FUNCTION_BLOCK FB_SelfTest IMPLEMENTS I_State
VAR_INPUT
	(* Pointer to the ATM Machine*)
	pATM_Machine	: POINTER TO FB_ATM_Machine;
END_VAR
VAR_OUTPUT
END_VAR
VAR
END_VAR

METHOD Cancel : BOOL
END_METHOD

METHOD Card_Ejected : BOOL
END_METHOD

METHOD Card_Inserted : BOOL
END_METHOD

PROPERTY Description : E_StateDescription
GET
Description := E_StateDescription.SelfTest;
END_GET
END_PROPERTY

METHOD Failure : BOOL
ADSLOGSTR(ADSLOG_MSGTYPE_LOG, 'System Test Fail, going to Out of Service', '');
pATM_Machine^.SetState(pATM_Machine^.OutOfServiceState);
END_METHOD

METHOD FB_Init : BOOL
VAR_INPUT
	(* if TRUE, the retain variables are initialized (warm start / cold start)*)
	bInitRetains	: BOOL;
	(* if TRUE, the instance afterwards gets moved into the copy code (online change)*)
	bInCopyCode	: BOOL;
	(* Pointer to the ATM Machine*)
	pATM_Machine	: POINTER TO FB_ATM_Machine;
END_VAR
THIS^.pATM_Machine := pATM_Machine;
END_METHOD

METHOD Op : BOOL
END_METHOD

METHOD Service : BOOL
END_METHOD

METHOD SystemTest_OK : BOOL
ADSLOGSTR(ADSLOG_MSGTYPE_LOG, 'System Test Pass, going to Idel', '');
pATM_Machine^.SetState(pATM_Machine^.IdleState);
END_METHOD

METHOD Turn_Off : BOOL
END_METHOD

METHOD Turn_On : BOOL
END_METHOD

END_FUNCTION_BLOCK

(* stored: Version 1.1.0.1, ProductVersion 3.1.4024.12
   POU FB_SelfTest: Id {bf530f68-0b58-001a-33dc-b8df2ba985a6}, SpecialFunc None
   Method Cancel: Id {ec583400-85a2-0439-03ef-a260f6c24af6}
   Method Card_Ejected: Id {241d4a32-2c17-08a8-2247-391cc109267f}
   Method Card_Inserted: Id {5dfbfab2-9050-0470-38d9-060a24f08e38}
   Property Description: Id {49a17546-5a47-0724-13e3-9f9fa5de2c14}
   Get Get: Id {25a9bd05-a407-0600-04e8-195918bff5e7}
   Method Failure: Id {02401ffa-9399-0930-3b2c-286699b159c8}
   Method FB_Init: Id {2ba494aa-bbc3-0f48-1716-5635010fb2f5}
   Method Op: Id {5a1a51f6-c898-05f2-1efd-750d1b4fe95c}
   Method Service: Id {b2723076-8d13-0f83-0514-3e1e79bed386}
   Method SystemTest_OK: Id {08998860-6ca0-06a3-2122-3d229dad0ca4}
   Method Turn_Off: Id {7e765441-1066-0b91-24ae-fa0271431b4f}
   Method Turn_On: Id {9a05e5cf-00c6-0992-1763-02b679060675} *)
